{attribute 'qualified_only'}
{attribute 'strict'}
TYPE MasterDevState :
(
	enum_member := 0
);
END_TYPE

(* stored: Version 1.1.0.1, ProductVersion 3.1.4024.11
   DUT MasterDevState: Id {73886f00-c457-4624-8eb2-cda6aaecdcb0} *)
